# EPICS substitutions: ek9000App/Db/EL3152.substitutions
file EL3152.template
{       pattern
        {
                TERMINAL,

        }
        {
        }
}
